Staubli VAL3: OnStart.pgx

public program OnStart(tool& x_tTool, trsf& x_trFrameOut)
begin
  //-----------------------------------------------------------------------
  //Header begin
  //Description of program
  //
  //Input parameters
  //  tool x_tTool:工具
  //  frame x_fFrame:参考坐标系

  //Output paramaters
  //  trsf x_trOffSetOut:新建坐标系的trsf值
  //
  //Example
  //  call OnStart(tool,frame,trTrsfSetOut)
  //History
  //  Creation : 2012-06-11 - PF.Zhong
  //Header end
  //-----------------------------------------------------------------------
  call init(x_tTool)
  if taskStatus("CheckModeFrame")!=-1
    taskKill("CheckModeFrame")
    wait(taskStatus("CheckModeFrame")==-1)
  endIf
  taskCreate "CheckModeFrame",15,CheckMode()
  call MainPage(x_trFrameOut)
end
